SUBAPPLICATION logiBUS_AI_Calibrate_IDA_OPC (* logiBUS_AI_IDA (Analog-Eingang) mit 2-Punkt-Kalibrierung (AR_CALIBRATE_SQ, INI-persistiert) auf VT-Zahlenfelder (Rohwert + kalibrierter Wert, je eigene CNumberVariable) + Bargraph (kalibriert) + 2 VT-Tasten (CO/CS) + OPC-UA (Rohwert DWORD + kalibrierter Wert REAL, generisch, ein Kanal) *)
  (* Standard: 61499-2; Description: Copyright (c) 2026 Meisterschulen am Ostbahnhof This program and the accompanying materials are made available under the terms of the Eclipse Public License 2.0 which is available at https://www.eclipse.org/legal/epl-2.0/ SPDX-License-Identifier: EPL-2.0 *)
  (* Version 1.0, 2026-08-31, Franz Höpfinger, Meisterschulen am Ostbahnhof, initial API and implementation and/or initial documentation - Kalibrierlogik nach Vorbild Uebung_028c3_AR.SUB, aber AR_CALIBRATE_SQ (korrigierte Offset-Formel, ECC-erzwungene CO-vor-CS-Reihenfolge) statt AR_CALIBRATE *)
  PACKAGE MyLib::sys;
  IMPORT isobus::UT::Q::const::IDs::ID_NULL;
  IMPORT logiBUS::io::AI::logiBUS_AI;
  IMPORT logiBUS::io::AI::logiBUS_AI_S;
  IMPORT logiBUS::utils::conversion::phys::NumericObjectPool_S;
  IMPORT isobus::UT::io::Button::ButtonActivationCode::BT_PRESSED_LATCHED;
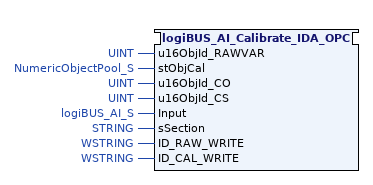
  VAR_INPUT
    u16ObjId_RAWVAR : UINT := ID_NULL; (* Object ID CNumberVariable (Rohwert 0-4095, unkalibriert, reine Diagnose-Anzeige) *)
    stObjCal : logiBUS::utils::conversion::phys::NumericObjectPool_S := (u16ObjId := ID_NULL, r32Scale := 1.0, i32Offset := 0, u8Decimals := 1); (* Object ID + Scale/Offset/Decimals CNumberVariable (kalibrierter Wert, eigene, unabhaengige CNumberVariable) *)
    u16ObjId_CO : UINT := ID_NULL; (* Object ID Taste 'CO' (Kalibrier-Nullpunkt: Referenz 1 anlegen, dann druecken) *)
    u16ObjId_CS : UINT := ID_NULL; (* Object ID Taste 'CS' (Kalibrier-Spanne: Referenz 2 anlegen, dann druecken - erst nach CO moeglich) *)
    Input : logiBUS::io::AI::logiBUS_AI_S := logiBUS_AI::Invalid; (* Identify the Input AnalogInput_I1..I8 *)
    sSection : STRING; (* INI-Sektionsname fuer OFFSET/SCALE-Persistenz - pro Kanal eindeutig (z.B. 'AI_Calibrate_I1'), sonst kollidieren die Kanaele in settings.ini *)
    ID_RAW_WRITE : WSTRING; (* Rohwert-Ruckmelde-Adresse (DWORD 0-4095, ACTION=PUBLISH) *)
    ID_CAL_WRITE : WSTRING; (* Kalibrierter-Wert-Ruckmelde-Adresse (REAL, ACTION=PUBLISH) *)
  END_VAR
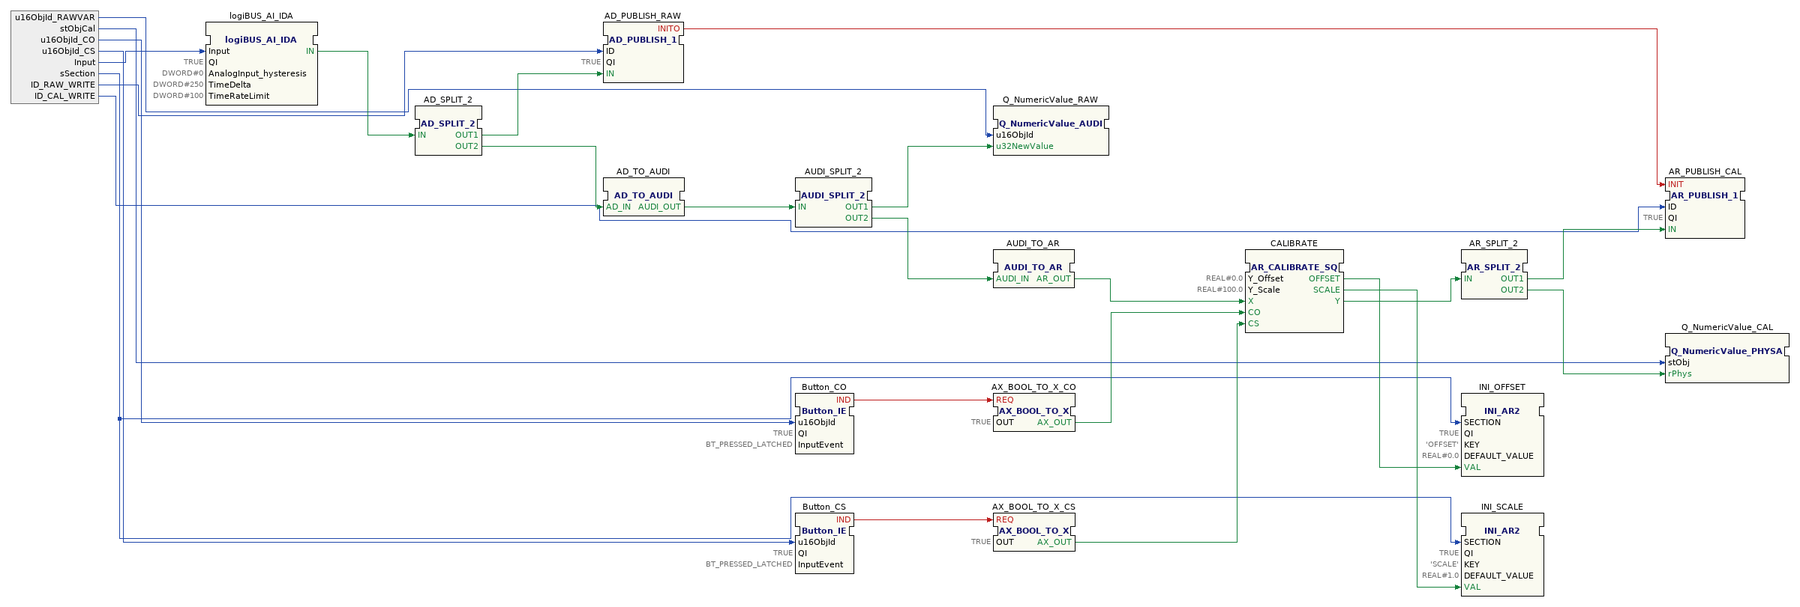
  FBS
    logiBUS_AI_IDA : logiBUS::io::AI::logiBUS_AI_IDA(QI := TRUE, AnalogInput_hysteresis := DWORD#0, TimeDelta := DWORD#250, TimeRateLimit := DWORD#100);
    AD_SPLIT_2 : adapter::events::unidirectional::AD_SPLIT_2;
    AD_PUBLISH_RAW : adapter::net::AD_PUBLISH_1(QI := TRUE);
    AD_TO_AUDI : adapter::conversion::unidirectional::AD_TO_AUDI;
    AUDI_SPLIT_2 : adapter::events::unidirectional::AUDI_SPLIT_2;
    Q_NumericValue_RAW : isobus::UT::Q::Q_NumericValue_AUDI;
    AUDI_TO_AR : adapter::conversion::unidirectional::AUDI_TO_AR;
    CALIBRATE : adapter::Engineering::measurements::AR_CALIBRATE_SQ(Y_Offset := REAL#0.0, Y_Scale := REAL#100.0);
    Button_CO : isobus::UT::io::Button::Button_IE(QI := TRUE, InputEvent := BT_PRESSED_LATCHED);
    Button_CS : isobus::UT::io::Button::Button_IE(QI := TRUE, InputEvent := BT_PRESSED_LATCHED);
    AX_BOOL_TO_X_CO : adapter::conversion::unidirectional::AX_BOOL_TO_X(OUT := TRUE);
    AX_BOOL_TO_X_CS : adapter::conversion::unidirectional::AX_BOOL_TO_X(OUT := TRUE);
    INI_OFFSET : eclipse4diac::storage::INI_AR2(QI := TRUE, KEY := 'OFFSET', DEFAULT_VALUE := REAL#0.0);
    INI_SCALE : eclipse4diac::storage::INI_AR2(QI := TRUE, KEY := 'SCALE', DEFAULT_VALUE := REAL#1.0);
    AR_SPLIT_2 : adapter::events::unidirectional::AR_SPLIT_2;
    AR_PUBLISH_CAL : adapter::net::AR_PUBLISH_1(QI := TRUE);
    Q_NumericValue_CAL : isobus::UT::Q::Q_NumericValue_PHYSA;
  END_FBS
  EVENT_CONNECTIONS
    AD_PUBLISH_RAW.INITO TO AR_PUBLISH_CAL.INIT;
    Button_CO.IND TO AX_BOOL_TO_X_CO.REQ;
    Button_CS.IND TO AX_BOOL_TO_X_CS.REQ;
  END_CONNECTIONS
  DATA_CONNECTIONS
    Input TO logiBUS_AI_IDA.Input;
    u16ObjId_RAWVAR TO Q_NumericValue_RAW.u16ObjId;
    stObjCal TO Q_NumericValue_CAL.stObj;
    u16ObjId_CO TO Button_CO.u16ObjId;
    u16ObjId_CS TO Button_CS.u16ObjId;
    sSection TO INI_OFFSET.SECTION;
    sSection TO INI_SCALE.SECTION;
    ID_RAW_WRITE TO AD_PUBLISH_RAW.ID;
    ID_CAL_WRITE TO AR_PUBLISH_CAL.ID;
  END_CONNECTIONS
  ADAPTER_CONNECTIONS
    logiBUS_AI_IDA.IN TO AD_SPLIT_2.IN;
    AD_SPLIT_2.OUT1 TO AD_PUBLISH_RAW.IN;
    AD_SPLIT_2.OUT2 TO AD_TO_AUDI.AD_IN;
    AD_TO_AUDI.AUDI_OUT TO AUDI_SPLIT_2.IN;
    AUDI_SPLIT_2.OUT1 TO Q_NumericValue_RAW.u32NewValue;
    AUDI_SPLIT_2.OUT2 TO AUDI_TO_AR.AUDI_IN;
    AUDI_TO_AR.AR_OUT TO CALIBRATE.X;
    AX_BOOL_TO_X_CO.AX_OUT TO CALIBRATE.CO;
    AX_BOOL_TO_X_CS.AX_OUT TO CALIBRATE.CS;
    CALIBRATE.OFFSET TO INI_OFFSET.VAL;
    CALIBRATE.SCALE TO INI_SCALE.VAL;
    CALIBRATE.Y TO AR_SPLIT_2.IN;
    AR_SPLIT_2.OUT1 TO AR_PUBLISH_CAL.IN;
    AR_SPLIT_2.OUT2 TO Q_NumericValue_CAL.rPhys;
  END_CONNECTIONS
END_SUBAPPLICATION
